// TIA Portal V21 export
VAR_GLOBAL   // PLC tag table "KSD1"
   KSD1CrusherBtnStartRaw AT %I8.0 : Bool;
   KSD1CrusherBtnStopRaw AT %I8.1 : Bool;
   KSD1CrusherKeySwitchRaw AT %I8.2 : Bool;
   KSD1CrusherEmStopRaw AT %I8.3 : Bool;
   KSD1CrusherBtnResetRaw AT %I8.4 : Bool;
   KSD1CrusherBtnStartLuSRaw AT %I8.5 : Bool;
   KSD1CrusherBtnStopLuSRaw AT %I8.6 : Bool;
   KSD1PremoldingSwRaw AT %I8.7 : Bool;
   KSD1PrestartAlmFbRaw AT %I9.0 : Bool;
   KSD1CrusherEccentricTempRaw AT %IW144 : Int;
   KSD1CrusherOuterBearingTempRaw AT %IW146 : Int;
   KSD1CrusherInnerBearingTempRaw AT %IW148 : Int;
   KSD1DriveFrontBearingTempRaw AT %IW150 : Int;
   KSD1DriveRearBearingTempRaw AT %IW152 : Int;
   KSD1DriveWindingTempP1Raw AT %IW154 : Int;
   KSD1DriveWindingTempP2Raw AT %IW156 : Int;
   KSD1DriveWindingTempP3Raw AT %IW158 : Int;
   KSD1DriveCurrentRaw AT %IW160 : Int;
   KSD1SgStartRaw AT %Q12.0 : Bool;
   KSD1SgStopRaw AT %Q12.1 : Bool;
   KSD1PreStartAlmOnRaw AT %Q12.2 : Bool;
   KSD1FeedEnRaw AT %Q12.3 : Bool;
   KSD1LuSLocalModeSwitchRaw AT %I9.1 : Bool;
   KSD1LuSBtnStartRaw AT %I9.2 : Bool;
   KSD1LuSBtnStopRaw AT %I9.3 : Bool;
   KSD1LuSBtnResetRaw AT %I9.4 : Bool;
   KSD1OilPump1SelSwitchRaw AT %I9.5 : Bool;
   KSD1OilPump2SelSwitchRaw AT %I9.6 : Bool;
   KSD1OilPreparationSwitchRaw AT %I9.7 : Bool;
   KSD1ReturnOilFlowSwitchRaw AT %I12.0 : Bool;
   KSD1OilLevelMaxRaw AT %I12.1 : Bool;
   KSD1OilLevelMidRaw AT %I12.2 : Bool;
   KSD1OilLevelMinRaw AT %I12.3 : Bool;
   KSD1OilTempSwitchHighRaw AT %I12.4 : Bool;
   KSD1OilTempSwitchLowRaw AT %I12.5 : Bool;
   KSD1FbPump1Raw AT %I12.6 : Bool;
   KSD1FbPump2Raw AT %I12.7 : Bool;
   KSD1Pump1FaultRaw AT %I13.0 : Bool;
   KSD1Pump2FaultRaw AT %I13.1 : Bool;
   KSD1OilTempTankRaw AT %IW162 : Int;
   KSD1ReturnOilTempRaw AT %IW168 : Int;
   KSD1OilFlowRaw AT %IW170 : Int;
   KSD1InletWaterTemperatureRaw AT %IW172 : Int;
   KSD1OutletWaterTemperatureRaw AT %IW174 : Int;
   KSD1InletOilTemperatureRaw AT %IW176 : Int;
   KSD1InletOilPressureRaw AT %IW178 : Int;
   KSD1Pump1StartRaw AT %Q12.4 : Bool;
   KSD1Pump2StartRaw AT %Q12.5 : Bool;
   KSD1HeaterOnRaw AT %Q12.6 : Bool;
   KSD1WaterVlvOpenRaw AT %Q12.7 : Bool;
   KSD1OilToCoolerVlvRaw AT %Q13.0 : Bool;
   KSD1SgReadyRaw AT %Q13.2 : Bool;
   KSD1SgFbOnRaw AT %Q13.3 : Bool;
   KSD1SgFbOffRaw AT %Q13.4 : Bool;
END_VAR
